PROGRAM robotAutomation
VAR
END_VAR

    IF(missionCompleted=1)THEN          // Same as StopMovement??}
      CASE userCommand OF
		  1,2,3:
		  	robotdata.activeState:=TURN_ENDED;
		4,5:
		robotdata.activeState:=MOVE_ENDED;
	  END_CASE
      robot_state:=0;
      modeEnable:=0;
      userCommand:=0;
    
    ELSIF(robot_state=0)THEN
      CASE userCommand OF
        1:  
          robot_state:=1;
          AngPosCommand:=myfmod(idealAngle+90,360)-180;
          modeEnable:=1;
          robotdata.motion_status:=MOTION_ANGLE;
          xGoal:=PosFdbckX;
          yGoal:=PosFdbckY;      
         2:          //TURN LEFT
          robot_state:=2;
          AngPosCommand:=myfmod(idealAngle-90,360)-180;
          modeEnable:=2;
          robotdata.motion_status:=MOTION_ANGLE;
          xGoal:=PosFdbckX;
          yGoal:=PosFdbckY;
         3:          //TURN BACK
          robot_state:=3;
          AngPosCommand:=myfmod(idealAngle+180,360);
          IF (AngPosCommand = 270) THEN
			AngPosCommand := -90;
			END_IF
          modeEnable:=3;
          robotdata.motion_status:=MOTION_ANGLE;
          xGoal:=PosFdbckX;
          yGoal:=PosFdbckY;
            
        4:           //FORWARD   
          robot_state:=4;
          robotdata.motion_status:=MOTION_ONGOING;
          xStart:=ltrunc(PosFdbckX);
          yStart:=ltrunc(PosFdbckY);
          xGoal:=xStart+COS(idealAngle*PI/180) * forwardCommand;
          yGoal:=yStart+SIN(idealAngle*PI/180) * forwardCommand;
          IF (xGoal >= 7) THEN
			xGoal := 7;
			END_IF
          IF (xGoal <= 0) THEN
			xGoal := 0;
		END_IF
          IF (yGoal >= 8) THEN 
			yGoal := 8;
			END_IF
          IF (yGoal <= 0) THEN 
			yGoal := 0;
			END_IF

          modeEnable:=4;
          
        5: // BACKWARD
          robot_state:=5;
          robotdata.motion_status:=MOTION_ONGOING;
          xStart:=ltrunc(PosFdbckX);
          yStart:=ltrunc(PosFdbckY);
          xGoal:=xStart - COS(idealAngle*PI/180) * forwardCommand;
          yGoal:=yStart - SIN(idealAngle*PI/180) * forwardCommand;
          IF (xGoal >= 7) THEN xGoal := 7; END_IF
          IF (xGoal <= 0) THEN xGoal := 0; END_IF
          IF (yGoal >= 8) THEN yGoal := 8; END_IF
          IF (yGoal <= 0) THEN yGoal := 0; END_IF
			  
		

          modeEnable:=5;
          
      END_CASE
    END_IF

END_PROGRAM

(* stored: Version 1.1.0.1, ProductVersion 3.1.4024.12
   POU robotAutomation: Id {6456eaca-18d3-42e2-8456-0ca2bb59e4b8}, SpecialFunc None *)
